FUNCTION_BLOCK FB_Beleuchtung
VAR_INPUT
END_VAR
VAR_OUTPUT
END_VAR
VAR
	Hallenbeleuchtung: FB_System_BelHa;
	Aussenbeleuchtung: FB_System_BelAu;
END_VAR

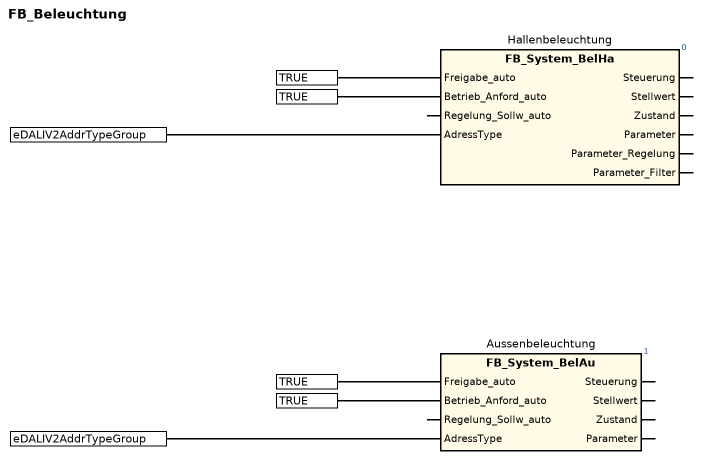
Hallenbeleuchtung(Freigabe_auto := TRUE, Betrieb_Anford_auto := TRUE, AdressType := eDALIV2AddrTypeGroup); // FB_System_BelHa
Aussenbeleuchtung(Freigabe_auto := TRUE, Betrieb_Anford_auto := TRUE, AdressType := eDALIV2AddrTypeGroup); // FB_System_BelAu

END_FUNCTION_BLOCK

(* stored: Version 1.1.0.1, ProductVersion 3.1.4024.9
   POU FB_Beleuchtung: Id {d91902a7-25f4-4ee4-a06d-89c71860e73f}, SpecialFunc None *)
